FUNCTION_BLOCK PackMlv3_StateModel
VAR_INPUT
	Cfg_RemoteCmdEnable: BOOL;
	Cmd_Mode: DINT;
	Cmd_Reset: BOOL;
	Cmd_Start: BOOL;
	Cmd_Stop: BOOL;
	Cmd_Hold: BOOL;
	Cmd_UnHold: BOOL;
	Cmd_Suspend: BOOL;
	Cmd_UnSuspend: BOOL;
	Cmd_Abort: BOOL;
	Cmd_Clear: BOOL;
	Cmd_StateComplete: BOOL;
	Inp_RemoteModeCmd: DINT;
	Inp_RemoteModeCmdChangeRequest: BOOL;
	Inp_RemoteStateCmd: DINT;
	Inp_RemoteStateCmdChangeRequest: BOOL;
END_VAR
VAR_OUTPUT
	Sts_StateCurrent: DINT;
	Sts_ModeCurrent: DINT;
	Sts_EnabledStates: DINT;
	Sts_ClearingEnabled: BOOL;
	Sts_StoppedEnabled: BOOL;
	Sts_StartingEnabled: BOOL;
	Sts_IdleEnabled: BOOL;
	Sts_SuspendedEnabled: BOOL;
	Sts_ExecuteEnabled: BOOL;
	Sts_StoppingEnabled: BOOL;
	Sts_AbortingEnabled: BOOL;
	Sts_AbortedEnabled: BOOL;
	Sts_HoldingEnabled: BOOL;
	Sts_HeldEnabled: BOOL;
	Sts_UnHoldingEnabled: BOOL;
	Sts_SuspendingEnabled: BOOL;
	Sts_UnSuspendingEnabled: BOOL;
	Sts_ResettingEnabled: BOOL;
	Sts_CompletingEnabled: BOOL;
	Sts_CompleteEnabled: BOOL;
	Sts_ModeChangeNotAllowed: BOOL;
	Sts_Clearing: BOOL;
	Sts_Stopped: BOOL;
	Sts_Starting: BOOL;
	Sts_Idle: BOOL;
	Sts_Suspended: BOOL;
	Sts_Execute: BOOL;
	Sts_Stopping: BOOL;
	Sts_Aborting: BOOL;
	Sts_Aborted: BOOL;
	Sts_Holding: BOOL;
	Sts_Held: BOOL;
	Sts_UnHolding: BOOL;
	Sts_Suspending: BOOL;
	Sts_UnSuspending: BOOL;
	Sts_Resetting: BOOL;
	Sts_Completing: BOOL;
	Sts_Complete: BOOL;
END_VAR
VAR_IN_OUT
	Cfg_ModeTransitions: ARRAY[0..31] OF DINT;
	Cfg_DisableStates: ARRAY[0..31] OF DINT;
	Cfg_ModeNames: ARRAY[0..31] OF STRING;
	Sts_StateCurrentName: STRING(255);	
	Sts_ModeCurrentName: STRING(255);	
END_VAR
VAR
	RemoteCmdChangeRequested: BOOL;
	ResetRemoteCmd: BOOL;
	StartRemoteCmd: BOOL;
	StopRemoteCmd: BOOL;
	HoldRemoteCmd: BOOL;
	UnholdRemoteCmd: BOOL;
	SuspendRemoteCmd: BOOL;
	UnSuspendRemoteCmd: BOOL;
	AbortRemoteCmd: BOOL;
	ClearRemoteCmd: BOOL;
	Cfg_DisableStatesCopy: DINT;
	StateComplete: BOOL;
	LocalClearing: BOOL;
	LocalStopped: BOOL;
	LocalStarting: BOOL;
	LocalExecute: BOOL;
	LocalCompleting: BOOL;
	LocalStopping: BOOL;
	LocalAborting: BOOL;
	LocalAborted: BOOL;
	LocalHolding: BOOL;
	LocalHeld: BOOL;
	LocalUnHolding: BOOL;
	LocalSuspending: BOOL;
	LocalSuspended: BOOL;
	LocalUnSuspending: BOOL;
	LocalResetting: BOOL;
	LocalIdle: BOOL;
	LocalComplete: BOOL;
	END_IFIF: INT;
	FS: BOOL;
END_VAR
VAR // added by the converter: edge detectors and wires of the graphical bodies
    _w1, _w2, _w3, _w4, _w5, _w6, _w7, _w8, _w9, _w10, _w11, _w12, _w13, _w14, _w15, _w16, _w17, _w18, _w19, _w20, _w21, _w22, _w23, _w24, _w25, _w26, _w27, _w28, _w29, _w30, _w31, _w32, _w33, _w34, _w35, _w36, _w37, _w38, _w39, _w40, _w41, _w42, _w43, _w44, _w45, _w46, _w47, _w48, _w49, _w50, _w51, _w52, _w53, _w54, _w55, _w56 : BOOL;
END_VAR


IF NOT FS THEN
	Sts_ModeCurrent:=1;
	Cmd_Mode:=1;
	StS_StateCurrent:=2;
    LocalClearing:=FALSE;
	LocalStopped:=TRUE;
	LocalStarting:=FALSE;
	LocalExecute:=FALSE;
	LocalCompleting:=FALSE;
	LocalStopping:=FALSE;
	LocalAborting:=FALSE;
	LocalAborted:=FALSE;
	LocalHolding:=FALSE;
	LocalHeld:=FALSE;
	LocalUnHolding:=FALSE;
	LocalSuspending:=FALSE;
	LocalSuspended:=FALSE;
	LocalUnSuspending:=FALSE;
	LocalResetting:=FALSE;
	LocalIdle:=FALSE;
	LocalComplete:=FALSE;
	FS:=TRUE;
END_IF
ACT();

IF Sts_StateCurrent=0 THEN
	IF RemoteCmdchangerequested AND inp_remoteModeCmd<>0 AND Inp_RemoteModeCmd>1 AND Inp_RemoteModeCmd<32 
	 AND Cfg_ModeTransitions[Sts_ModeCurrent].0 AND Cfg_ModeTransitions[Inp_RemoteModeCmd].0 THEN
		Sts_ModeCurrent:=Inp_RemoteModeCmd;
		Cmd_Mode:=Sts_ModeCurrent;
	END_IF
	IF Cmd_Mode<>Sts_ModeCurrent AND Cmd_Mode>1 AND Cmd_Mode<32 
	 AND Cfg_ModeTransitions[Sts_ModeCurrent].0 AND Cfg_ModeTransitions[Cmd_Mode].0 THEN	
		Sts_ModeCurrent:=Cmd_Mode;
	END_IF
	
END_IF
IF Sts_StateCurrent=1 THEN
	IF RemoteCmdchangerequested AND inp_remoteModeCmd<>0 AND Inp_RemoteModeCmd>1 AND Inp_RemoteModeCmd<32 
	 AND Cfg_ModeTransitions[Sts_ModeCurrent].1 AND Cfg_ModeTransitions[Inp_RemoteModeCmd].1 THEN
		Sts_ModeCurrent:=Inp_RemoteModeCmd;
		Cmd_Mode:=Sts_ModeCurrent;
	END_IF
	IF Cmd_Mode<>Sts_ModeCurrent AND Cmd_Mode>1 AND Cmd_Mode<32 
	 AND Cfg_ModeTransitions[Sts_ModeCurrent].1 AND Cfg_ModeTransitions[Cmd_Mode].1 THEN	
		Sts_ModeCurrent:=Cmd_Mode;
	END_IF
END_IF
IF Sts_StateCurrent=2 THEN
	IF RemoteCmdchangerequested AND inp_remoteModeCmd<>0 AND Inp_RemoteModeCmd>1 AND Inp_RemoteModeCmd<32 
	 AND Cfg_ModeTransitions[Sts_ModeCurrent].2 AND Cfg_ModeTransitions[Inp_RemoteModeCmd].2 THEN
		Sts_ModeCurrent:=Inp_RemoteModeCmd;
		Cmd_Mode:=Sts_ModeCurrent;
	END_IF
	IF Cmd_Mode<>Sts_ModeCurrent AND Cmd_Mode>1 AND Cmd_Mode<32 
	 AND Cfg_ModeTransitions[Sts_ModeCurrent].2 AND Cfg_ModeTransitions[Cmd_Mode].2 THEN	
		Sts_ModeCurrent:=Cmd_Mode;
	END_IF
END_IF
IF Sts_StateCurrent=3 THEN
	IF RemoteCmdchangerequested AND inp_remoteModeCmd<>0 AND Inp_RemoteModeCmd>1 AND Inp_RemoteModeCmd<32 
	 AND Cfg_ModeTransitions[Sts_ModeCurrent].3 AND Cfg_ModeTransitions[Inp_RemoteModeCmd].3 THEN
		Sts_ModeCurrent:=Inp_RemoteModeCmd;
		Cmd_Mode:=Sts_ModeCurrent;
	END_IF
	IF Cmd_Mode<>Sts_ModeCurrent AND Cmd_Mode>1 AND Cmd_Mode<32 
	 AND Cfg_ModeTransitions[Sts_ModeCurrent].3 AND Cfg_ModeTransitions[Cmd_Mode].3 THEN	
		Sts_ModeCurrent:=Cmd_Mode;
	END_IF
END_IF
IF Sts_StateCurrent=4 THEN
	IF RemoteCmdchangerequested AND inp_remoteModeCmd<>0 AND Inp_RemoteModeCmd>1 AND Inp_RemoteModeCmd<32 
	 AND Cfg_ModeTransitions[Sts_ModeCurrent].4 AND Cfg_ModeTransitions[Inp_RemoteModeCmd].4 THEN
		Sts_ModeCurrent:=Inp_RemoteModeCmd;
		Cmd_Mode:=Sts_ModeCurrent;
	END_IF
	IF Cmd_Mode<>Sts_ModeCurrent AND Cmd_Mode>1 AND Cmd_Mode<32 
	 AND Cfg_ModeTransitions[Sts_ModeCurrent].4 AND Cfg_ModeTransitions[Cmd_Mode].4 THEN	
		Sts_ModeCurrent:=Cmd_Mode;
	END_IF
END_IF
IF Sts_StateCurrent=5 THEN
	IF RemoteCmdchangerequested AND inp_remoteModeCmd<>0 AND Inp_RemoteModeCmd>1 AND Inp_RemoteModeCmd<32 
	 AND Cfg_ModeTransitions[Sts_ModeCurrent].5 AND Cfg_ModeTransitions[Inp_RemoteModeCmd].5 THEN
		Sts_ModeCurrent:=Inp_RemoteModeCmd;
		Cmd_Mode:=Sts_ModeCurrent;
	END_IF
	IF Cmd_Mode<>Sts_ModeCurrent AND Cmd_Mode>1 AND Cmd_Mode<32 
	 AND Cfg_ModeTransitions[Sts_ModeCurrent].5 AND Cfg_ModeTransitions[Cmd_Mode].5 THEN	
		Sts_ModeCurrent:=Cmd_Mode;
	END_IF
END_IF
IF Sts_StateCurrent=6 THEN
	IF RemoteCmdchangerequested AND inp_remoteModeCmd<>0 AND Inp_RemoteModeCmd>1 AND Inp_RemoteModeCmd<32 
	 AND Cfg_ModeTransitions[Sts_ModeCurrent].6 AND Cfg_ModeTransitions[Inp_RemoteModeCmd].6 THEN
		Sts_ModeCurrent:=Inp_RemoteModeCmd;
		Cmd_Mode:=Sts_ModeCurrent;
	END_IF
	IF Cmd_Mode<>Sts_ModeCurrent AND Cmd_Mode>1 AND Cmd_Mode<32 
	 AND Cfg_ModeTransitions[Sts_ModeCurrent].6 AND Cfg_ModeTransitions[Cmd_Mode].6 THEN	
		Sts_ModeCurrent:=Cmd_Mode;
	END_IF
END_IF
IF Sts_StateCurrent=7 THEN
	IF RemoteCmdchangerequested AND inp_remoteModeCmd<>0 AND Inp_RemoteModeCmd>1 AND Inp_RemoteModeCmd<32 
	 AND Cfg_ModeTransitions[Sts_ModeCurrent].7 AND Cfg_ModeTransitions[Inp_RemoteModeCmd].7 THEN
		Sts_ModeCurrent:=Inp_RemoteModeCmd;
		Cmd_Mode:=Sts_ModeCurrent;
	END_IF
	IF Cmd_Mode<>Sts_ModeCurrent AND Cmd_Mode>1 AND Cmd_Mode<32 
	 AND Cfg_ModeTransitions[Sts_ModeCurrent].7 AND Cfg_ModeTransitions[Cmd_Mode].7 THEN	
		Sts_ModeCurrent:=Cmd_Mode;
	END_IF
END_IF
IF Sts_StateCurrent=8 THEN
	IF RemoteCmdchangerequested AND inp_remoteModeCmd<>0 AND Inp_RemoteModeCmd>1 AND Inp_RemoteModeCmd<32 
	 AND Cfg_ModeTransitions[Sts_ModeCurrent].8 AND Cfg_ModeTransitions[Inp_RemoteModeCmd].8 THEN
		Sts_ModeCurrent:=Inp_RemoteModeCmd;
		Cmd_Mode:=Sts_ModeCurrent;
	END_IF
	IF Cmd_Mode<>Sts_ModeCurrent AND Cmd_Mode>1 AND Cmd_Mode<32 
	 AND Cfg_ModeTransitions[Sts_ModeCurrent].8 AND Cfg_ModeTransitions[Cmd_Mode].8 THEN	
		Sts_ModeCurrent:=Cmd_Mode;
	END_IF
END_IF
IF Sts_StateCurrent=9 THEN
	IF RemoteCmdchangerequested AND inp_remoteModeCmd<>0 AND Inp_RemoteModeCmd>1 AND Inp_RemoteModeCmd<32 
	 AND Cfg_ModeTransitions[Sts_ModeCurrent].9 AND Cfg_ModeTransitions[Inp_RemoteModeCmd].9 THEN
		Sts_ModeCurrent:=Inp_RemoteModeCmd;
		Cmd_Mode:=Sts_ModeCurrent;
	END_IF
	IF Cmd_Mode<>Sts_ModeCurrent AND Cmd_Mode>1 AND Cmd_Mode<32 
	 AND Cfg_ModeTransitions[Sts_ModeCurrent].9 AND Cfg_ModeTransitions[Cmd_Mode].9 THEN	
		Sts_ModeCurrent:=Cmd_Mode;
	END_IF
END_IF
IF Sts_StateCurrent=10 THEN
	IF RemoteCmdchangerequested AND inp_remoteModeCmd<>0 AND Inp_RemoteModeCmd>1 AND Inp_RemoteModeCmd<32 
	 AND Cfg_ModeTransitions[Sts_ModeCurrent].10 AND Cfg_ModeTransitions[Inp_RemoteModeCmd].10 THEN
		Sts_ModeCurrent:=Inp_RemoteModeCmd;
		Cmd_Mode:=Sts_ModeCurrent;
	END_IF
	IF Cmd_Mode<>Sts_ModeCurrent AND Cmd_Mode>1 AND Cmd_Mode<32 
	 AND Cfg_ModeTransitions[Sts_ModeCurrent].10 AND Cfg_ModeTransitions[Cmd_Mode].10 THEN	
		Sts_ModeCurrent:=Cmd_Mode;
	END_IF
END_IF
IF Sts_StateCurrent=11 THEN
	IF RemoteCmdchangerequested AND inp_remoteModeCmd<>0 AND Inp_RemoteModeCmd>1 AND Inp_RemoteModeCmd<32 
	 AND Cfg_ModeTransitions[Sts_ModeCurrent].11 AND Cfg_ModeTransitions[Inp_RemoteModeCmd].11 THEN
		Sts_ModeCurrent:=Inp_RemoteModeCmd;
		Cmd_Mode:=Sts_ModeCurrent;
	END_IF
	IF Cmd_Mode<>Sts_ModeCurrent AND Cmd_Mode>1 AND Cmd_Mode<32 
	 AND Cfg_ModeTransitions[Sts_ModeCurrent].11 AND Cfg_ModeTransitions[Cmd_Mode].11 THEN	
		Sts_ModeCurrent:=Cmd_Mode;
	END_IF
END_IF
IF Sts_StateCurrent=12 THEN
	IF RemoteCmdchangerequested AND inp_remoteModeCmd<>0 AND Inp_RemoteModeCmd>1 AND Inp_RemoteModeCmd<32 
	 AND Cfg_ModeTransitions[Sts_ModeCurrent].12 AND Cfg_ModeTransitions[Inp_RemoteModeCmd].12 THEN
		Sts_ModeCurrent:=Inp_RemoteModeCmd;
		Cmd_Mode:=Sts_ModeCurrent;
	END_IF
	IF Cmd_Mode<>Sts_ModeCurrent AND Cmd_Mode>1 AND Cmd_Mode<32 
	 AND Cfg_ModeTransitions[Sts_ModeCurrent].12 AND Cfg_ModeTransitions[Cmd_Mode].12 THEN	
		Sts_ModeCurrent:=Cmd_Mode;
	END_IF
END_IF
IF Sts_StateCurrent=13 THEN
	IF RemoteCmdchangerequested AND inp_remoteModeCmd<>0 AND Inp_RemoteModeCmd>1 AND Inp_RemoteModeCmd<32 
	 AND Cfg_ModeTransitions[Sts_ModeCurrent].13 AND Cfg_ModeTransitions[Inp_RemoteModeCmd].13 THEN
		Sts_ModeCurrent:=Inp_RemoteModeCmd;
		Cmd_Mode:=Sts_ModeCurrent;
	END_IF
	IF Cmd_Mode<>Sts_ModeCurrent AND Cmd_Mode>1 AND Cmd_Mode<32 
	 AND Cfg_ModeTransitions[Sts_ModeCurrent].13 AND Cfg_ModeTransitions[Cmd_Mode].13 THEN	
		Sts_ModeCurrent:=Cmd_Mode;
	END_IF
END_IF
IF Sts_StateCurrent=14 THEN
	IF RemoteCmdchangerequested AND inp_remoteModeCmd<>0 AND Inp_RemoteModeCmd>1 AND Inp_RemoteModeCmd<32 
	 AND Cfg_ModeTransitions[Sts_ModeCurrent].14 AND Cfg_ModeTransitions[Inp_RemoteModeCmd].14 THEN
		Sts_ModeCurrent:=Inp_RemoteModeCmd;
		Cmd_Mode:=Sts_ModeCurrent;
	END_IF
	IF Cmd_Mode<>Sts_ModeCurrent AND Cmd_Mode>1 AND Cmd_Mode<32 
	 AND Cfg_ModeTransitions[Sts_ModeCurrent].14 AND Cfg_ModeTransitions[Cmd_Mode].14 THEN	
		Sts_ModeCurrent:=Cmd_Mode;
	END_IF
END_IF
IF Sts_StateCurrent=15 THEN
	IF RemoteCmdchangerequested AND inp_remoteModeCmd<>0 AND Inp_RemoteModeCmd>1 AND Inp_RemoteModeCmd<32 
	 AND Cfg_ModeTransitions[Sts_ModeCurrent].15 AND Cfg_ModeTransitions[Inp_RemoteModeCmd].15 THEN
		Sts_ModeCurrent:=Inp_RemoteModeCmd;
		Cmd_Mode:=Sts_ModeCurrent;
	END_IF
	IF Cmd_Mode<>Sts_ModeCurrent AND Cmd_Mode>1 AND Cmd_Mode<32 
	 AND Cfg_ModeTransitions[Sts_ModeCurrent].15 AND Cfg_ModeTransitions[Cmd_Mode].15 THEN	
		Sts_ModeCurrent:=Cmd_Mode;
	END_IF
END_IF
IF Sts_StateCurrent=16 THEN
	IF RemoteCmdchangerequested AND inp_remoteModeCmd<>0 AND Inp_RemoteModeCmd>1 AND Inp_RemoteModeCmd<32 
	 AND Cfg_ModeTransitions[Sts_ModeCurrent].16 AND Cfg_ModeTransitions[Inp_RemoteModeCmd].16 THEN
		Sts_ModeCurrent:=Inp_RemoteModeCmd;
		Cmd_Mode:=Sts_ModeCurrent;
	END_IF
	IF Cmd_Mode<>Sts_ModeCurrent AND Cmd_Mode>1 AND Cmd_Mode<32 
	 AND Cfg_ModeTransitions[Sts_ModeCurrent].16 AND Cfg_ModeTransitions[Cmd_Mode].16 THEN	
		Sts_ModeCurrent:=Cmd_Mode;
	END_IF
END_IF	
IF Sts_StateCurrent=17 THEN
	IF RemoteCmdchangerequested AND inp_remoteModeCmd<>0 AND Inp_RemoteModeCmd>1 AND Inp_RemoteModeCmd<32 
	 AND Cfg_ModeTransitions[Sts_ModeCurrent].17 AND Cfg_ModeTransitions[Inp_RemoteModeCmd].17 THEN
		Sts_ModeCurrent:=Inp_RemoteModeCmd;
		Cmd_Mode:=Sts_ModeCurrent;
	END_IF
	IF Cmd_Mode<>Sts_ModeCurrent AND Cmd_Mode>1 AND Cmd_Mode<32 
	 AND Cfg_ModeTransitions[Sts_ModeCurrent].17 AND Cfg_ModeTransitions[Cmd_Mode].17 THEN	
		Sts_ModeCurrent:=Cmd_Mode;
	END_IF
END_IF
IF Sts_StateCurrent=18 THEN
	IF RemoteCmdchangerequested AND inp_remoteModeCmd<>0 AND Inp_RemoteModeCmd>1 AND Inp_RemoteModeCmd<32 
	 AND Cfg_ModeTransitions[Sts_ModeCurrent].18 AND Cfg_ModeTransitions[Inp_RemoteModeCmd].18 THEN
		Sts_ModeCurrent:=Inp_RemoteModeCmd;
		Cmd_Mode:=Sts_ModeCurrent;
	END_IF
	IF Cmd_Mode<>Sts_ModeCurrent AND Cmd_Mode>1 AND Cmd_Mode<32 
	 AND Cfg_ModeTransitions[Sts_ModeCurrent].18 AND Cfg_ModeTransitions[Cmd_Mode].18 THEN	
		Sts_ModeCurrent:=Cmd_Mode;
	END_IF
END_IF
IF Sts_StateCurrent=19 THEN
	IF RemoteCmdchangerequested AND inp_remoteModeCmd<>0 AND Inp_RemoteModeCmd>1 AND Inp_RemoteModeCmd<32 
	 AND Cfg_ModeTransitions[Sts_ModeCurrent].19 AND Cfg_ModeTransitions[Inp_RemoteModeCmd].19 THEN
		Sts_ModeCurrent:=Inp_RemoteModeCmd;
		Cmd_Mode:=Sts_ModeCurrent;
	END_IF
	IF Cmd_Mode<>Sts_ModeCurrent AND Cmd_Mode>1 AND Cmd_Mode<32 
	 AND Cfg_ModeTransitions[Sts_ModeCurrent].19 AND Cfg_ModeTransitions[Cmd_Mode].19 THEN	
		Sts_ModeCurrent:=Cmd_Mode;
	END_IF
END_IF
IF Sts_StateCurrent=20 THEN
	IF RemoteCmdchangerequested AND inp_remoteModeCmd<>0 AND Inp_RemoteModeCmd>1 AND Inp_RemoteModeCmd<32 
	 AND Cfg_ModeTransitions[Sts_ModeCurrent].20 AND Cfg_ModeTransitions[Inp_RemoteModeCmd].20 THEN
		Sts_ModeCurrent:=Inp_RemoteModeCmd;
		Cmd_Mode:=Sts_ModeCurrent;
	END_IF
	IF Cmd_Mode<>Sts_ModeCurrent AND Cmd_Mode>1 AND Cmd_Mode<32 
	 AND Cfg_ModeTransitions[Sts_ModeCurrent].20 AND Cfg_ModeTransitions[Cmd_Mode].20 THEN	
		Sts_ModeCurrent:=Cmd_Mode;
	END_IF
END_IF
IF Sts_StateCurrent=21 THEN
	IF RemoteCmdchangerequested AND inp_remoteModeCmd<>0 AND Inp_RemoteModeCmd>1 AND Inp_RemoteModeCmd<32 
	 AND Cfg_ModeTransitions[Sts_ModeCurrent].21 AND Cfg_ModeTransitions[Inp_RemoteModeCmd].21 THEN
		Sts_ModeCurrent:=Inp_RemoteModeCmd;
		Cmd_Mode:=Sts_ModeCurrent;
	END_IF
	IF Cmd_Mode<>Sts_ModeCurrent AND Cmd_Mode>1 AND Cmd_Mode<32 
	 AND Cfg_ModeTransitions[Sts_ModeCurrent].21 AND Cfg_ModeTransitions[Cmd_Mode].21 THEN	
		Sts_ModeCurrent:=Cmd_Mode;
	END_IF
END_IF
IF Sts_StateCurrent=22 THEN
	IF RemoteCmdchangerequested AND inp_remoteModeCmd<>0 AND Inp_RemoteModeCmd>1 AND Inp_RemoteModeCmd<32 
	 AND Cfg_ModeTransitions[Sts_ModeCurrent].22 AND Cfg_ModeTransitions[Inp_RemoteModeCmd].22 THEN
		Sts_ModeCurrent:=Inp_RemoteModeCmd;
		Cmd_Mode:=Sts_ModeCurrent;
	END_IF
	IF Cmd_Mode<>Sts_ModeCurrent AND Cmd_Mode>1 AND Cmd_Mode<32 
	 AND Cfg_ModeTransitions[Sts_ModeCurrent].22 AND Cfg_ModeTransitions[Cmd_Mode].22 THEN	
		Sts_ModeCurrent:=Cmd_Mode;
	END_IF
END_IF
IF Sts_StateCurrent=23 THEN
	IF RemoteCmdchangerequested AND inp_remoteModeCmd<>0 AND Inp_RemoteModeCmd>1 AND Inp_RemoteModeCmd<32 
	 AND Cfg_ModeTransitions[Sts_ModeCurrent].23 AND Cfg_ModeTransitions[Inp_RemoteModeCmd].23 THEN
		Sts_ModeCurrent:=Inp_RemoteModeCmd;
		Cmd_Mode:=Sts_ModeCurrent;
	END_IF
	IF Cmd_Mode<>Sts_ModeCurrent AND Cmd_Mode>1 AND Cmd_Mode<32 
	 AND Cfg_ModeTransitions[Sts_ModeCurrent].23 AND Cfg_ModeTransitions[Cmd_Mode].23 THEN	
		Sts_ModeCurrent:=Cmd_Mode;
	END_IF
END_IF
IF Sts_StateCurrent=24 THEN
	IF RemoteCmdchangerequested AND inp_remoteModeCmd<>0 AND Inp_RemoteModeCmd>1 AND Inp_RemoteModeCmd<32 
	 AND Cfg_ModeTransitions[Sts_ModeCurrent].24 AND Cfg_ModeTransitions[Inp_RemoteModeCmd].24 THEN
		Sts_ModeCurrent:=Inp_RemoteModeCmd;
		Cmd_Mode:=Sts_ModeCurrent;
	END_IF
	IF Cmd_Mode<>Sts_ModeCurrent AND Cmd_Mode>1 AND Cmd_Mode<32 
	 AND Cfg_ModeTransitions[Sts_ModeCurrent].24 AND Cfg_ModeTransitions[Cmd_Mode].24 THEN	
		Sts_ModeCurrent:=Cmd_Mode;
	END_IF
END_IF
IF Sts_StateCurrent=25 THEN
	IF RemoteCmdchangerequested AND inp_remoteModeCmd<>0 AND Inp_RemoteModeCmd>1 AND Inp_RemoteModeCmd<32 
	 AND Cfg_ModeTransitions[Sts_ModeCurrent].25 AND Cfg_ModeTransitions[Inp_RemoteModeCmd].25 THEN
		Sts_ModeCurrent:=Inp_RemoteModeCmd;
		Cmd_Mode:=Sts_ModeCurrent;
	END_IF
	IF Cmd_Mode<>Sts_ModeCurrent AND Cmd_Mode>1 AND Cmd_Mode<32 
	 AND Cfg_ModeTransitions[Sts_ModeCurrent].25 AND Cfg_ModeTransitions[Cmd_Mode].25 THEN	
		Sts_ModeCurrent:=Cmd_Mode;
	END_IF
END_IF
IF Sts_StateCurrent=26 THEN
	IF RemoteCmdchangerequested AND inp_remoteModeCmd<>0 AND Inp_RemoteModeCmd>1 AND Inp_RemoteModeCmd<32 
	 AND Cfg_ModeTransitions[Sts_ModeCurrent].26 AND Cfg_ModeTransitions[Inp_RemoteModeCmd].26 THEN
		Sts_ModeCurrent:=Inp_RemoteModeCmd;
		Cmd_Mode:=Sts_ModeCurrent;
	END_IF
	IF Cmd_Mode<>Sts_ModeCurrent AND Cmd_Mode>1 AND Cmd_Mode<32 
	 AND Cfg_ModeTransitions[Sts_ModeCurrent].26 AND Cfg_ModeTransitions[Cmd_Mode].26 THEN	
		Sts_ModeCurrent:=Cmd_Mode;
	END_IF
END_IF
IF Sts_StateCurrent=27 THEN
	IF RemoteCmdchangerequested AND inp_remoteModeCmd<>0 AND Inp_RemoteModeCmd>1 AND Inp_RemoteModeCmd<32 
	 AND Cfg_ModeTransitions[Sts_ModeCurrent].27 AND Cfg_ModeTransitions[Inp_RemoteModeCmd].27 THEN
		Sts_ModeCurrent:=Inp_RemoteModeCmd;
		Cmd_Mode:=Sts_ModeCurrent;
	END_IF
	IF Cmd_Mode<>Sts_ModeCurrent AND Cmd_Mode>1 AND Cmd_Mode<32 
	 AND Cfg_ModeTransitions[Sts_ModeCurrent].27 AND Cfg_ModeTransitions[Cmd_Mode].27 THEN	
		Sts_ModeCurrent:=Cmd_Mode;
	END_IF
END_IF
IF Sts_StateCurrent=28 THEN
	IF RemoteCmdchangerequested AND inp_remoteModeCmd<>0 AND Inp_RemoteModeCmd>1 AND Inp_RemoteModeCmd<32 
	 AND Cfg_ModeTransitions[Sts_ModeCurrent].28 AND Cfg_ModeTransitions[Inp_RemoteModeCmd].28 THEN
		Sts_ModeCurrent:=Inp_RemoteModeCmd;
		Cmd_Mode:=Sts_ModeCurrent;
	END_IF
	IF Cmd_Mode<>Sts_ModeCurrent AND Cmd_Mode>1 AND Cmd_Mode<32 
	 AND Cfg_ModeTransitions[Sts_ModeCurrent].28 AND Cfg_ModeTransitions[Cmd_Mode].28 THEN	
		Sts_ModeCurrent:=Cmd_Mode;
	END_IF
END_IF
IF Sts_StateCurrent=29 THEN
	IF RemoteCmdchangerequested AND inp_remoteModeCmd<>0 AND Inp_RemoteModeCmd>1 AND Inp_RemoteModeCmd<32 
	 AND Cfg_ModeTransitions[Sts_ModeCurrent].29 AND Cfg_ModeTransitions[Inp_RemoteModeCmd].29 THEN
		Sts_ModeCurrent:=Inp_RemoteModeCmd;
		Cmd_Mode:=Sts_ModeCurrent;
	END_IF
	IF Cmd_Mode<>Sts_ModeCurrent AND Cmd_Mode>1 AND Cmd_Mode<32 
	 AND Cfg_ModeTransitions[Sts_ModeCurrent].29 AND Cfg_ModeTransitions[Cmd_Mode].29 THEN	
		Sts_ModeCurrent:=Cmd_Mode;
	END_IF
END_IF
IF Sts_StateCurrent=30 THEN
	IF RemoteCmdchangerequested AND inp_remoteModeCmd<>0 AND Inp_RemoteModeCmd>1 AND Inp_RemoteModeCmd<32 
	 AND Cfg_ModeTransitions[Sts_ModeCurrent].30 AND Cfg_ModeTransitions[Inp_RemoteModeCmd].30 THEN
		Sts_ModeCurrent:=Inp_RemoteModeCmd;
		Cmd_Mode:=Sts_ModeCurrent;
	END_IF
	IF Cmd_Mode<>Sts_ModeCurrent AND Cmd_Mode>1 AND Cmd_Mode<32 
	 AND Cfg_ModeTransitions[Sts_ModeCurrent].30 AND Cfg_ModeTransitions[Cmd_Mode].30 THEN	
		Sts_ModeCurrent:=Cmd_Mode;
	END_IF
END_IF
IF Sts_StateCurrent=31 THEN
	IF RemoteCmdchangerequested AND inp_remoteModeCmd<>0 AND Inp_RemoteModeCmd>1 AND Inp_RemoteModeCmd<32 
	 AND Cfg_ModeTransitions[Sts_ModeCurrent].31 AND Cfg_ModeTransitions[Inp_RemoteModeCmd].31 THEN
		Sts_ModeCurrent:=Inp_RemoteModeCmd;
		Cmd_Mode:=Sts_ModeCurrent;
	END_IF
	IF Cmd_Mode<>Sts_ModeCurrent AND Cmd_Mode>1 AND Cmd_Mode<32 
	 AND Cfg_ModeTransitions[Sts_ModeCurrent].31 AND Cfg_ModeTransitions[Cmd_Mode].31 THEN	
		Sts_ModeCurrent:=Cmd_Mode;
	END_IF
END_IF

ACTION ACT:
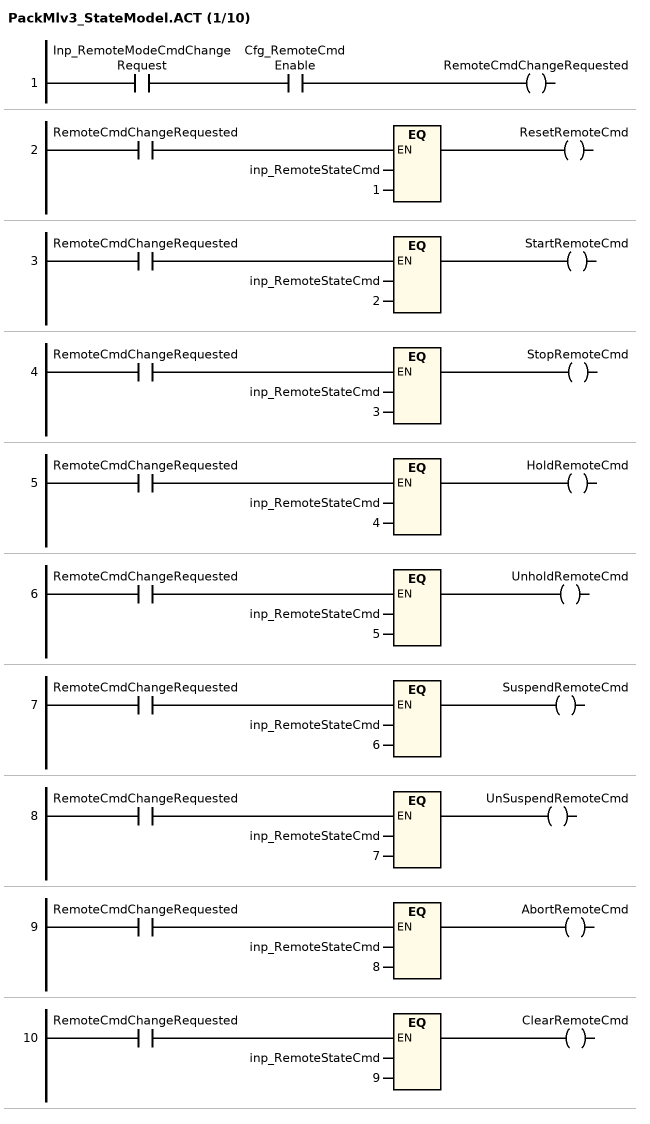
// NETWORK 1
RemoteCmdChangeRequested := Inp_RemoteModeCmdChangeRequest AND Cfg_RemoteCmdEnable;

// NETWORK 2
ResetRemoteCmd := RemoteCmdChangeRequested AND inp_RemoteStateCmd = 1;

// NETWORK 3
StartRemoteCmd := RemoteCmdChangeRequested AND inp_RemoteStateCmd = 2;

// NETWORK 4
StopRemoteCmd := RemoteCmdChangeRequested AND inp_RemoteStateCmd = 3;

// NETWORK 5
HoldRemoteCmd := RemoteCmdChangeRequested AND inp_RemoteStateCmd = 4;

// NETWORK 6
UnholdRemoteCmd := RemoteCmdChangeRequested AND inp_RemoteStateCmd = 5;

// NETWORK 7
SuspendRemoteCmd := RemoteCmdChangeRequested AND inp_RemoteStateCmd = 6;

// NETWORK 8
UnSuspendRemoteCmd := RemoteCmdChangeRequested AND inp_RemoteStateCmd = 7;

// NETWORK 9
AbortRemoteCmd := RemoteCmdChangeRequested AND inp_RemoteStateCmd = 8;

// NETWORK 10
ClearRemoteCmd := RemoteCmdChangeRequested AND inp_RemoteStateCmd = 9;

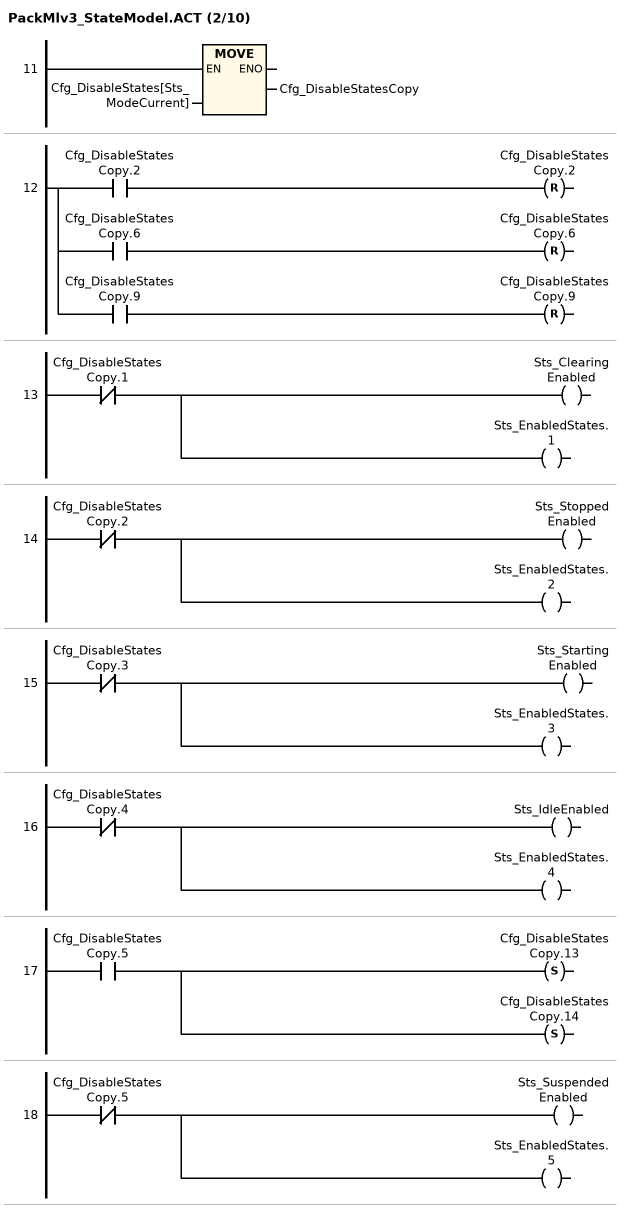
// NETWORK 11
Cfg_DisableStatesCopy := Cfg_DisableStates[Sts_ModeCurrent];

// NETWORK 12
Cfg_DisableStatesCopy.2 R= Cfg_DisableStatesCopy.2;
Cfg_DisableStatesCopy.6 R= Cfg_DisableStatesCopy.6;
Cfg_DisableStatesCopy.9 R= Cfg_DisableStatesCopy.9;

// NETWORK 13
_w1 := NOT Cfg_DisableStatesCopy.1;
Sts_ClearingEnabled := _w1;
Sts_EnabledStates.1 := _w1;

// NETWORK 14
_w2 := NOT Cfg_DisableStatesCopy.2;
Sts_StoppedEnabled := _w2;
Sts_EnabledStates.2 := _w2;

// NETWORK 15
_w3 := NOT Cfg_DisableStatesCopy.3;
Sts_StartingEnabled := _w3;
Sts_EnabledStates.3 := _w3;

// NETWORK 16
_w4 := NOT Cfg_DisableStatesCopy.4;
Sts_IdleEnabled := _w4;
Sts_EnabledStates.4 := _w4;

// NETWORK 17
_w5 := Cfg_DisableStatesCopy.5;
Cfg_DisableStatesCopy.13 S= _w5;
Cfg_DisableStatesCopy.14 S= _w5;

// NETWORK 18
_w6 := NOT Cfg_DisableStatesCopy.5;
Sts_SuspendedEnabled := _w6;
Sts_EnabledStates.5 := _w6;

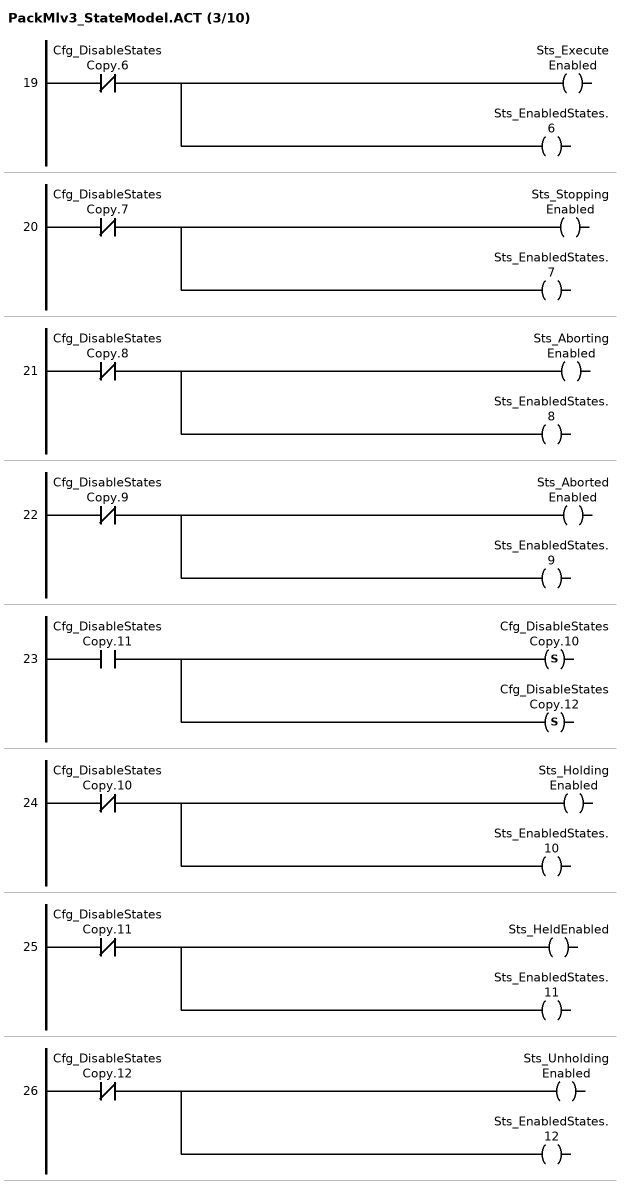
// NETWORK 19
_w7 := NOT Cfg_DisableStatesCopy.6;
Sts_ExecuteEnabled := _w7;
Sts_EnabledStates.6 := _w7;

// NETWORK 20
_w8 := NOT Cfg_DisableStatesCopy.7;
Sts_StoppingEnabled := _w8;
Sts_EnabledStates.7 := _w8;

// NETWORK 21
_w9 := NOT Cfg_DisableStatesCopy.8;
Sts_AbortingEnabled := _w9;
Sts_EnabledStates.8 := _w9;

// NETWORK 22
_w10 := NOT Cfg_DisableStatesCopy.9;
Sts_AbortedEnabled := _w10;
Sts_EnabledStates.9 := _w10;

// NETWORK 23
_w11 := Cfg_DisableStatesCopy.11;
Cfg_DisableStatesCopy.10 S= _w11;
Cfg_DisableStatesCopy.12 S= _w11;

// NETWORK 24
_w12 := NOT Cfg_DisableStatesCopy.10;
Sts_HoldingEnabled := _w12;
Sts_EnabledStates.10 := _w12;

// NETWORK 25
_w13 := NOT Cfg_DisableStatesCopy.11;
Sts_HeldEnabled := _w13;
Sts_EnabledStates.11 := _w13;

// NETWORK 26
_w14 := NOT Cfg_DisableStatesCopy.12;
Sts_UnholdingEnabled := _w14;
Sts_EnabledStates.12 := _w14;

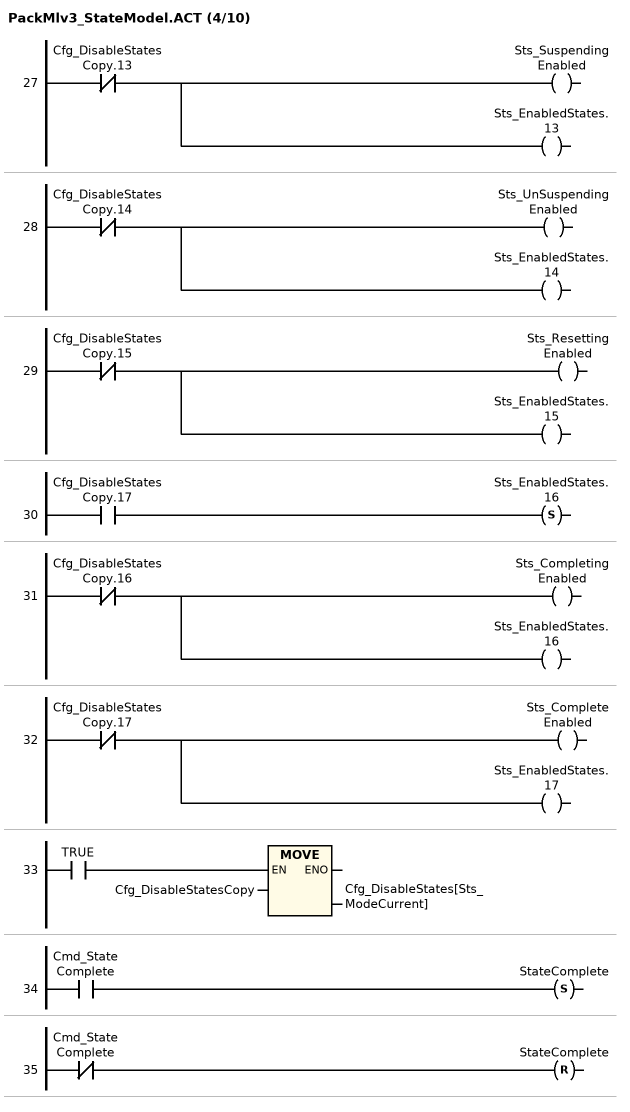
// NETWORK 27
_w15 := NOT Cfg_DisableStatesCopy.13;
Sts_SuspendingEnabled := _w15;
Sts_EnabledStates.13 := _w15;

// NETWORK 28
_w16 := NOT Cfg_DisableStatesCopy.14;
Sts_UnSuspendingEnabled := _w16;
Sts_EnabledStates.14 := _w16;

// NETWORK 29
_w17 := NOT Cfg_DisableStatesCopy.15;
Sts_ResettingEnabled := _w17;
Sts_EnabledStates.15 := _w17;

// NETWORK 30
Sts_EnabledStates.16 S= Cfg_DisableStatesCopy.17;

// NETWORK 31
_w18 := NOT Cfg_DisableStatesCopy.16;
Sts_CompletingEnabled := _w18;
Sts_EnabledStates.16 := _w18;

// NETWORK 32
_w19 := NOT Cfg_DisableStatesCopy.17;
Sts_CompleteEnabled := _w19;
Sts_EnabledStates.17 := _w19;

// NETWORK 33
Cfg_DisableStates[Sts_ModeCurrent] := Cfg_DisableStatesCopy;

// NETWORK 34
StateComplete S= Cmd_StateComplete;

// NETWORK 35
StateComplete R= NOT Cmd_StateComplete;

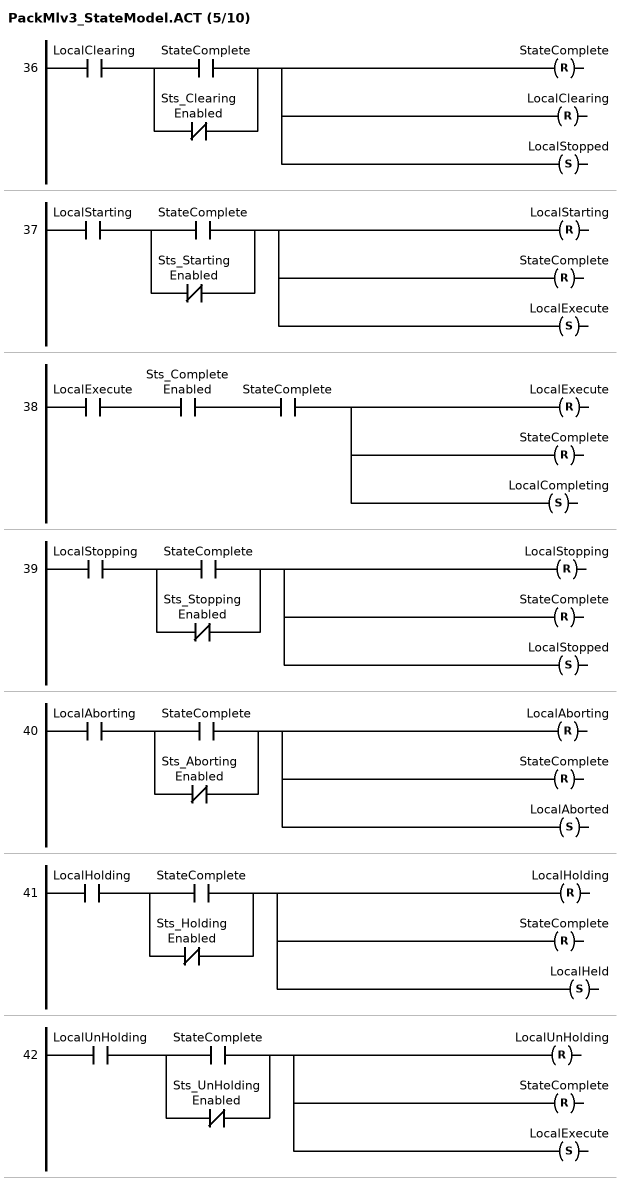
// NETWORK 36
_w20 := LocalClearing AND (StateComplete OR NOT Sts_ClearingEnabled);
StateComplete R= _w20;
LocalClearing R= _w20;
LocalStopped S= _w20;

// NETWORK 37
_w21 := LocalStarting AND (StateComplete OR NOT Sts_StartingEnabled);
LocalStarting R= _w21;
StateComplete R= _w21;
LocalExecute S= _w21;

// NETWORK 38
_w22 := LocalExecute AND Sts_CompleteEnabled AND StateComplete;
LocalExecute R= _w22;
StateComplete R= _w22;
LocalCompleting S= _w22;

// NETWORK 39
_w23 := LocalStopping AND (StateComplete OR NOT Sts_StoppingEnabled);
LocalStopping R= _w23;
StateComplete R= _w23;
LocalStopped S= _w23;

// NETWORK 40
_w24 := LocalAborting AND (StateComplete OR NOT Sts_AbortingEnabled);
LocalAborting R= _w24;
StateComplete R= _w24;
LocalAborted S= _w24;

// NETWORK 41
_w25 := LocalHolding AND (StateComplete OR NOT Sts_HoldingEnabled);
LocalHolding R= _w25;
StateComplete R= _w25;
LocalHeld S= _w25;

// NETWORK 42
_w26 := LocalUnHolding AND (StateComplete OR NOT Sts_UnHoldingEnabled);
LocalUnHolding R= _w26;
StateComplete R= _w26;
LocalExecute S= _w26;

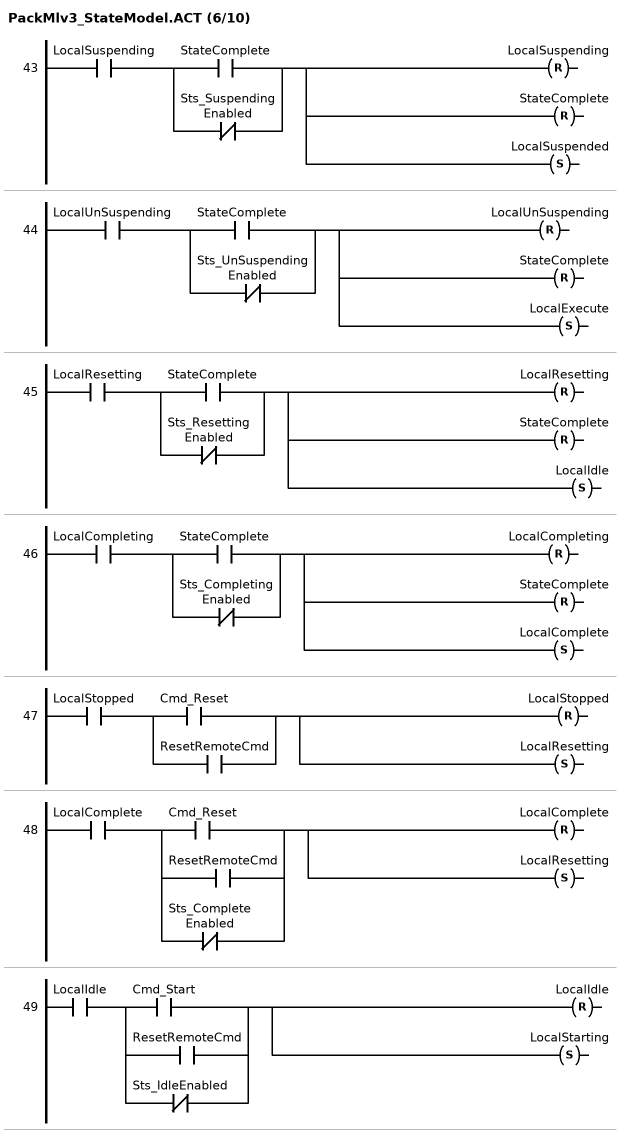
// NETWORK 43
_w27 := LocalSuspending AND (StateComplete OR NOT Sts_SuspendingEnabled);
LocalSuspending R= _w27;
StateComplete R= _w27;
LocalSuspended S= _w27;

// NETWORK 44
_w28 := LocalUnSuspending AND (StateComplete OR NOT Sts_UnSuspendingEnabled);
LocalUnSuspending R= _w28;
StateComplete R= _w28;
LocalExecute S= _w28;

// NETWORK 45
_w29 := LocalResetting AND (StateComplete OR NOT Sts_ResettingEnabled);
LocalResetting R= _w29;
StateComplete R= _w29;
LocalIdle S= _w29;

// NETWORK 46
_w30 := LocalCompleting AND (StateComplete OR NOT Sts_CompletingEnabled);
LocalCompleting R= _w30;
StateComplete R= _w30;
LocalComplete S= _w30;

// NETWORK 47
_w31 := LocalStopped AND (Cmd_Reset OR ResetRemoteCmd);
LocalStopped R= _w31;
LocalResetting S= _w31;

// NETWORK 48
_w32 := LocalComplete AND (Cmd_Reset OR ResetRemoteCmd OR NOT Sts_CompleteEnabled);
LocalComplete R= _w32;
LocalResetting S= _w32;

// NETWORK 49
_w33 := LocalIdle AND (Cmd_Start OR ResetRemoteCmd OR NOT Sts_IdleEnabled);
LocalIdle R= _w33;
LocalStarting S= _w33;

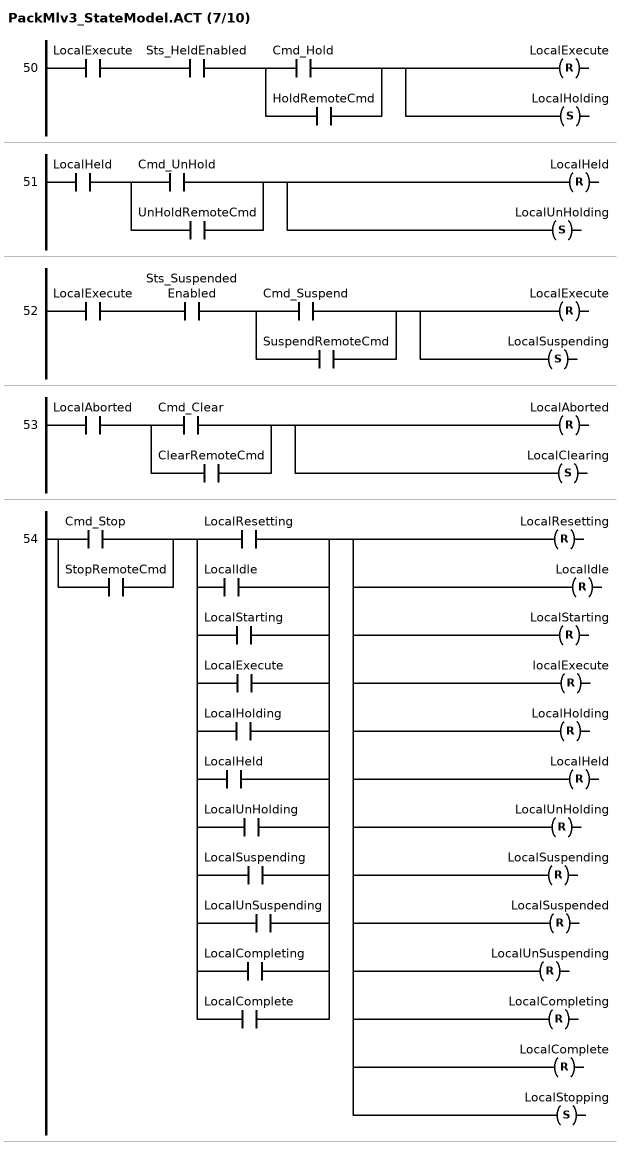
// NETWORK 50
_w34 := LocalExecute AND Sts_HeldEnabled AND (Cmd_Hold OR HoldRemoteCmd);
LocalExecute R= _w34;
LocalHolding S= _w34;

// NETWORK 51
_w35 := LocalHeld AND (Cmd_UnHold OR UnHoldRemoteCmd);
LocalHeld R= _w35;
LocalUnHolding S= _w35;

// NETWORK 52
_w36 := LocalExecute AND Sts_SuspendedEnabled AND (Cmd_Suspend OR SuspendRemoteCmd);
LocalExecute R= _w36;
LocalSuspending S= _w36;

// NETWORK 53
_w37 := LocalAborted AND (Cmd_Clear OR ClearRemoteCmd);
LocalAborted R= _w37;
LocalClearing S= _w37;

// NETWORK 54
_w38 := (Cmd_Stop OR StopRemoteCmd) AND (LocalResetting OR LocalIdle OR LocalStarting OR LocalExecute OR LocalHolding OR LocalHeld OR LocalUnHolding OR LocalSuspending OR LocalUnSuspending OR LocalCompleting OR LocalComplete);
LocalResetting R= _w38;
LocalIdle R= _w38;
LocalStarting R= _w38;
localExecute R= _w38;
LocalHolding R= _w38;
LocalHeld R= _w38;
LocalUnHolding R= _w38;
LocalSuspending R= _w38;
LocalSuspended R= _w38;
LocalUnSuspending R= _w38;
LocalCompleting R= _w38;
LocalComplete R= _w38;
LocalStopping S= _w38;

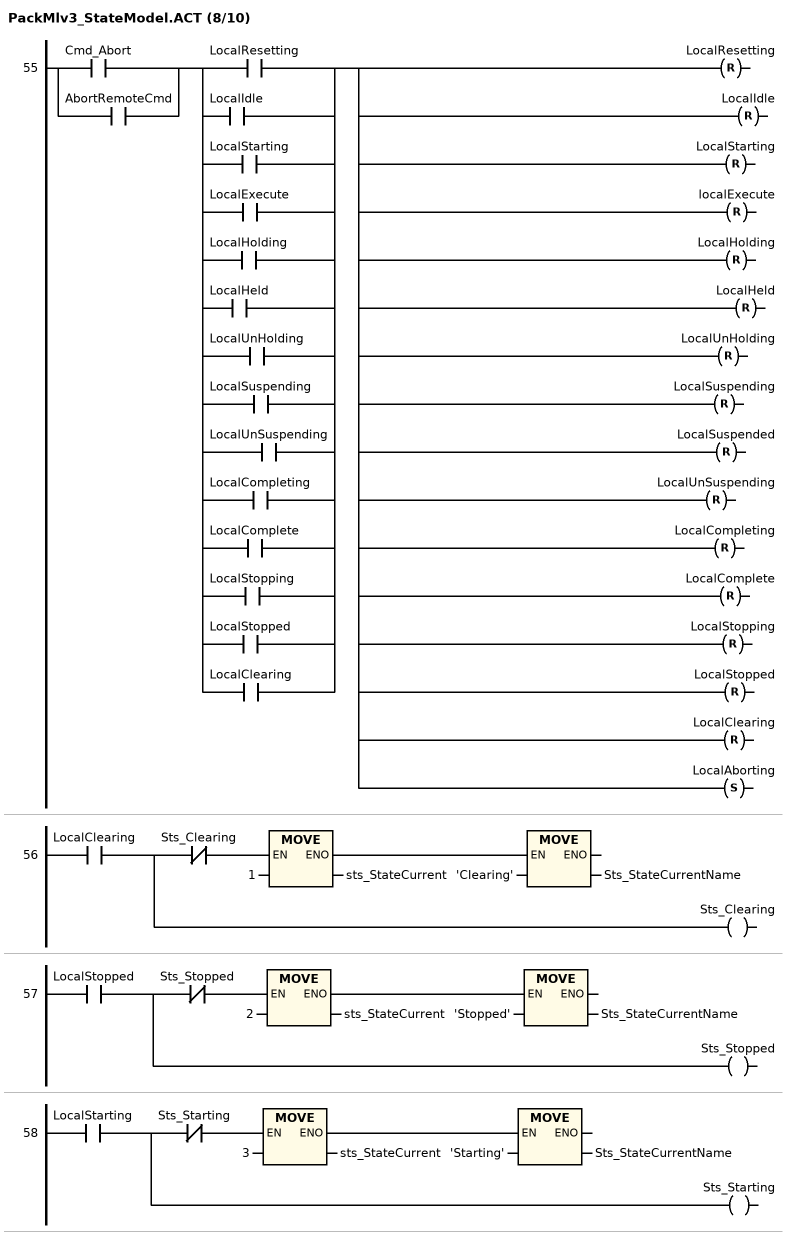
// NETWORK 55
_w39 := (Cmd_Abort OR AbortRemoteCmd) AND (LocalResetting OR LocalIdle OR LocalStarting OR LocalExecute OR LocalHolding OR LocalHeld OR LocalUnHolding OR LocalSuspending OR LocalUnSuspending OR LocalCompleting OR LocalComplete OR LocalStopping OR LocalStopped OR LocalClearing);
LocalResetting R= _w39;
LocalIdle R= _w39;
LocalStarting R= _w39;
localExecute R= _w39;
LocalHolding R= _w39;
LocalHeld R= _w39;
LocalUnHolding R= _w39;
LocalSuspending R= _w39;
LocalSuspended R= _w39;
LocalUnSuspending R= _w39;
LocalCompleting R= _w39;
LocalComplete R= _w39;
LocalStopping R= _w39;
LocalStopped R= _w39;
LocalClearing R= _w39;
LocalAborting S= _w39;

// NETWORK 56
_w40 := LocalClearing AND NOT Sts_Clearing;
IF _w40 THEN sts_StateCurrent := 1; END_IF
IF _w40 THEN Sts_StateCurrentName := 'Clearing'; END_IF
Sts_Clearing := LocalClearing;

// NETWORK 57
_w41 := LocalStopped AND NOT Sts_Stopped;
IF _w41 THEN sts_StateCurrent := 2; END_IF
IF _w41 THEN Sts_StateCurrentName := 'Stopped'; END_IF
Sts_Stopped := LocalStopped;

// NETWORK 58
_w42 := LocalStarting AND NOT Sts_Starting;
IF _w42 THEN sts_StateCurrent := 3; END_IF
IF _w42 THEN Sts_StateCurrentName := 'Starting'; END_IF
Sts_Starting := LocalStarting;

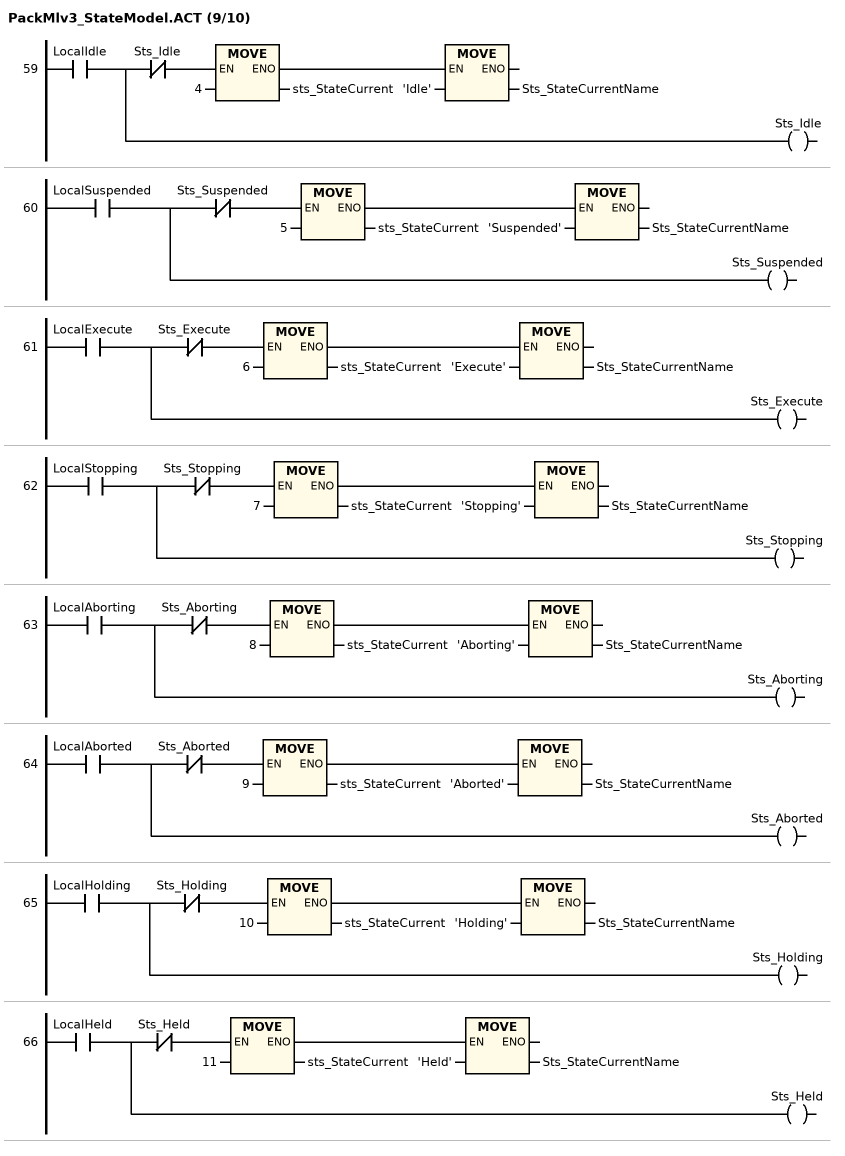
// NETWORK 59
_w43 := LocalIdle AND NOT Sts_Idle;
IF _w43 THEN sts_StateCurrent := 4; END_IF
IF _w43 THEN Sts_StateCurrentName := 'Idle'; END_IF
Sts_Idle := LocalIdle;

// NETWORK 60
_w44 := LocalSuspended AND NOT Sts_Suspended;
IF _w44 THEN sts_StateCurrent := 5; END_IF
IF _w44 THEN Sts_StateCurrentName := 'Suspended'; END_IF
Sts_Suspended := LocalSuspended;

// NETWORK 61
_w45 := LocalExecute AND NOT Sts_Execute;
IF _w45 THEN sts_StateCurrent := 6; END_IF
IF _w45 THEN Sts_StateCurrentName := 'Execute'; END_IF
Sts_Execute := LocalExecute;

// NETWORK 62
_w46 := LocalStopping AND NOT Sts_Stopping;
IF _w46 THEN sts_StateCurrent := 7; END_IF
IF _w46 THEN Sts_StateCurrentName := 'Stopping'; END_IF
Sts_Stopping := LocalStopping;

// NETWORK 63
_w47 := LocalAborting AND NOT Sts_Aborting;
IF _w47 THEN sts_StateCurrent := 8; END_IF
IF _w47 THEN Sts_StateCurrentName := 'Aborting'; END_IF
Sts_Aborting := LocalAborting;

// NETWORK 64
_w48 := LocalAborted AND NOT Sts_Aborted;
IF _w48 THEN sts_StateCurrent := 9; END_IF
IF _w48 THEN Sts_StateCurrentName := 'Aborted'; END_IF
Sts_Aborted := LocalAborted;

// NETWORK 65
_w49 := LocalHolding AND NOT Sts_Holding;
IF _w49 THEN sts_StateCurrent := 10; END_IF
IF _w49 THEN Sts_StateCurrentName := 'Holding'; END_IF
Sts_Holding := LocalHolding;

// NETWORK 66
_w50 := LocalHeld AND NOT Sts_Held;
IF _w50 THEN sts_StateCurrent := 11; END_IF
IF _w50 THEN Sts_StateCurrentName := 'Held'; END_IF
Sts_Held := LocalHeld;

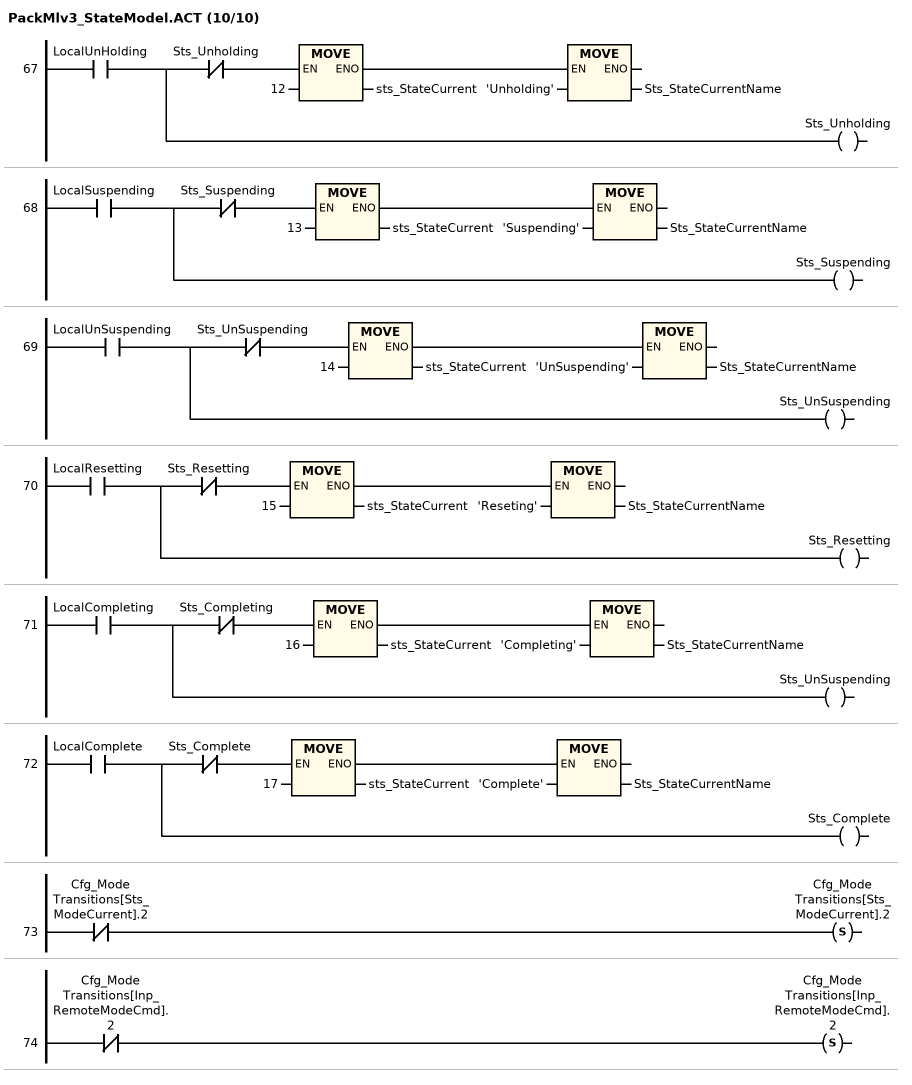
// NETWORK 67
_w51 := LocalUnHolding AND NOT Sts_Unholding;
IF _w51 THEN sts_StateCurrent := 12; END_IF
IF _w51 THEN Sts_StateCurrentName := 'Unholding'; END_IF
Sts_Unholding := LocalUnHolding;

// NETWORK 68
_w52 := LocalSuspending AND NOT Sts_Suspending;
IF _w52 THEN sts_StateCurrent := 13; END_IF
IF _w52 THEN Sts_StateCurrentName := 'Suspending'; END_IF
Sts_Suspending := LocalSuspending;

// NETWORK 69
_w53 := LocalUnSuspending AND NOT Sts_UnSuspending;
IF _w53 THEN sts_StateCurrent := 14; END_IF
IF _w53 THEN Sts_StateCurrentName := 'UnSuspending'; END_IF
Sts_UnSuspending := LocalUnSuspending;

// NETWORK 70
_w54 := LocalResetting AND NOT Sts_Resetting;
IF _w54 THEN sts_StateCurrent := 15; END_IF
IF _w54 THEN Sts_StateCurrentName := 'Reseting'; END_IF
Sts_Resetting := LocalResetting;

// NETWORK 71
_w55 := LocalCompleting AND NOT Sts_Completing;
IF _w55 THEN sts_StateCurrent := 16; END_IF
IF _w55 THEN Sts_StateCurrentName := 'Completing'; END_IF
Sts_UnSuspending := LocalCompleting;

// NETWORK 72
_w56 := LocalComplete AND NOT Sts_Complete;
IF _w56 THEN sts_StateCurrent := 17; END_IF
IF _w56 THEN Sts_StateCurrentName := 'Complete'; END_IF
Sts_Complete := LocalComplete;

// NETWORK 73
Cfg_ModeTransitions[Sts_ModeCurrent].2 S= NOT Cfg_ModeTransitions[Sts_ModeCurrent].2;

// NETWORK 74
Cfg_ModeTransitions[Inp_RemoteModeCmd].2 S= NOT Cfg_ModeTransitions[Inp_RemoteModeCmd].2;
END_ACTION

END_FUNCTION_BLOCK

(* stored: Version 1.1.0.1, ProductVersion 3.1.4022.16
   POU PackMlv3_StateModel: Id {a03b2f76-9b56-4455-9de0-8d6b561c1964}, SpecialFunc None
   Action ACT: Id {a806867d-1664-4b16-a553-c5c35f44f6e9} *)
